// TIA Portal V19 export
TYPE "LEXCHANGETRAY_typeSr1000ProfinetTelegram_unstableReadStatusBits"
// stored: Access Published
   STRUCT
      statusByte : Byte;
      unstable : Bool;
      matchingLevelUnstable : Bool;
      isoIec15415Unstable : Bool;
      aimdpmUnstable : Bool;
      saeAs9132Unstable : Bool;
   END_STRUCT;
END_TYPE
